fbSlamutak(
    X1 := GVL_R2.Nivaa,
    X2 := GVL_Rest.siSivState,
    XE := XE,
    SivValve1BCL := PS00_VP01.BCL,
    SivValve2BCL := PS00_VP02.BCL,
    SivValve3BCL := PS00_VP03.BCL,
    SivValve4BCL := PS00_VP04.BCL,
    ReactorValveBCL := PS02_VP01.BCL,
    ReactorValveBCH := PS02_VP01.BCH,
    PTI := GVL_Rest.Uttaksintervall,
    PTMT := GVL_Rest.MaxGangtidSlam,
    PRAntattSlamNivaa := GVL_Rest.AntattSlamNivaa);
GVL_Rest.PulseCoutner := fbSlamutak.Y;
// -------------------------------------------------------------------------------------------------------------------------------- OUTPUTS --------------------------------------------------------------------------------------------------------------------------------
// Reaktor Slamventil
// INPUTS
PS02_VP01(XGH := Sim1.BCH, XGL := Sim1.BCL, XH := fbSlamutak.YHReactorValve, XL := fbSlamutak.YLReactorValve); // SBV
Sim1(X := PS02_VP01.Y); // fbValveSim
// OUTPUTS
GVL_Outputs.PS02_VP01_Y := PS02_VP01.Y;
GVL_R2.PS02_VP01_YF := PS02_VP01.YF;
// Sivebed1
// INPUTS
PS00_VP01(XGH := Sim2.BCH, XGL := Sim2.BCL, XH := fbSlamutak.YHSivbed1Valve, XL := fbSlamutak.YLSivbed1Valve); // SBV
Sim2(X := PS00_VP01.Y); // fbValveSim
// OUTPUTS
GVL_R2.PS00_VP01_Y := PS00_VP01.Y;
GVL_R2.PS00_VP01_YF := PS00_VP01.YF;
// Sivebed2
// INPUTS
PS00_VP02(XGH := Sim3.BCH, XGL := Sim3.BCL, XH := fbSlamutak.YHSivbed2Valve, XL := fbSlamutak.YLSivbed2Valve); // SBV
Sim3(X := PS00_VP02.Y); // fbValveSim
// OUTPUTS
GVL_R2.PS00_VP02_Y := PS00_VP02.Y;
GVL_R2.PS00_VP02_YF := PS00_VP02.YF;
// Sivebed3
// INPUTS
PS00_VP03(XGH := Sim4.BCH, XGL := Sim4.BCL, XH := fbSlamutak.YHSivbed3Valve, XL := fbSlamutak.YLSivbed3Valve); // SBV
Sim4(X := PS00_VP03.Y); // fbValveSim
// OUTPUTS
GVL_R2.PS00_VP03_Y := PS00_VP03.Y;
GVL_R2.PS00_VP03_YF := PS00_VP03.YF;
// Sivebed4
// INPUTS
PS00_VP04(XGH := Sim4.BCH, XGL := Sim4.BCL, XH := fbSlamutak.YHSivbed4Valve, XL := fbSlamutak.YLSivbed4Valve); // SBV
Sim4(X := PS00_VP04.Y); // fbValveSim
// OUTPUTS
GVL_R2.PS00_VP04_Y := PS00_VP04.Y;
GVL_R2.PS00_VP04_YF := PS00_VP04.YF;

END_FUNCTION_BLOCK

// Device/Application/Simulation/Analog_I
FUNCTION_BLOCK Analog_I
VAR_INPUT
	FillLevelR	: REAL;
END_VAR
VAR_IN_OUT
	FillLevelInt	: INT;
END_VAR
VAR
	L1: LIN_TRAFO;
	L2: LIN_TRAFO;
//END_VAR
//VAR_TEMP
	Kast	: BOOL;
	temp		: REAL;
	FillV	: REAL;
END_VAR

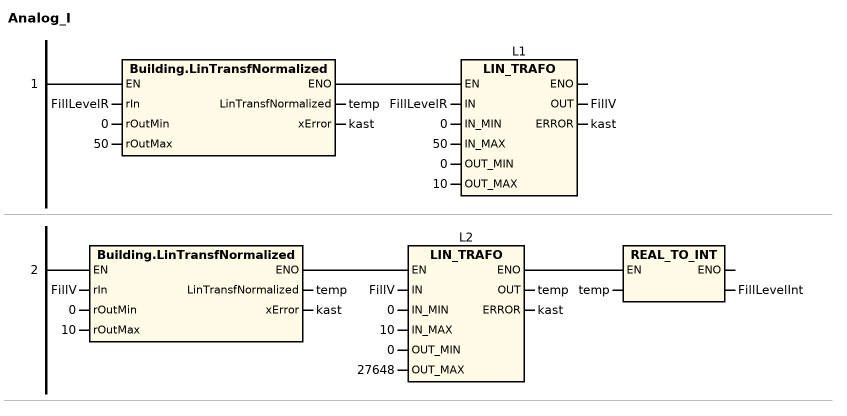
// NETWORK 1
temp := Building.LinTransfNormalized(rIn := FillLevelR, rOutMin := 0, rOutMax := 50, xError => kast);
L1(IN := FillLevelR, IN_MIN := 0, IN_MAX := 50, OUT_MIN := 0, OUT_MAX := 10, OUT => FillV, ERROR => kast); // LIN_TRAFO

// NETWORK 2
temp := Building.LinTransfNormalized(rIn := FillV, rOutMin := 0, rOutMax := 10, xError => kast);
L2(IN := FillV, IN_MIN := 0, IN_MAX := 10, OUT_MIN := 0, OUT_MAX := 27648, OUT => temp, ERROR => kast); // LIN_TRAFO
FillLevelInt := REAL_TO_INT(temp);

END_FUNCTION_BLOCK

// Device/Application/Simulation/Analog_O
FUNCTION_BLOCK Analog_O
VAR_INPUT
	PLC_Output	: INT;
END_VAR
VAR_IN_OUT
	Flow		: REAL;
END_VAR
VAR
	L1: LIN_TRAFO;
	L2: LIN_TRAFO;
//END_VAR
//VAR_TEMP
	Kast	: BOOL;
	temp		: REAL;
	PlcV	: REAL;
END_VAR

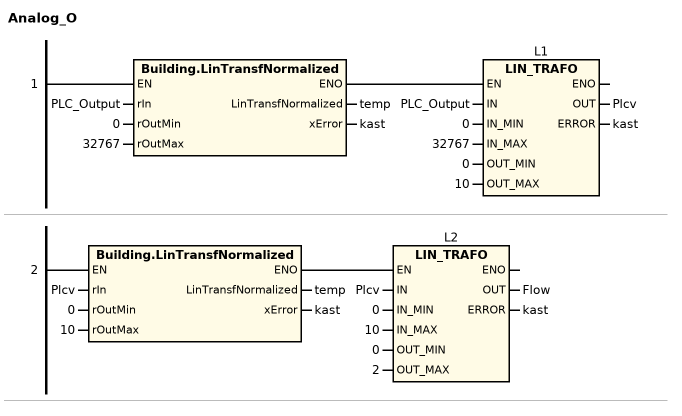
// NETWORK 1
temp := Building.LinTransfNormalized(rIn := PLC_Output, rOutMin := 0, rOutMax := 32767, xError => kast);
L1(IN := PLC_Output, IN_MIN := 0, IN_MAX := 32767, OUT_MIN := 0, OUT_MAX := 10, OUT => Plcv, ERROR => kast); // LIN_TRAFO

// NETWORK 2
temp := Building.LinTransfNormalized(rIn := Plcv, rOutMin := 0, rOutMax := 10, xError => kast);
L2(IN := Plcv, IN_MIN := 0, IN_MAX := 10, OUT_MIN := 0, OUT_MAX := 2, OUT => Flow, ERROR => kast); // LIN_TRAFO

END_FUNCTION_BLOCK

// Device/Application/Simulation/fbTankTest
FUNCTION_BLOCK fbTankTest
VAR_INPUT
	
	Start			: BOOL;	// Start av simulasjon

	StartNivaa		: REAL;	// Ved start av simulasjon kor mykje % er i tanken
	FillPerSekund	: INT;	// Tilrenning mot tank
	
	TankHoyde		: REAL;	// Dimensjonering av tank
	TankBreidde		: REAL;	// Dimensjonering av tank
	TankLengde		: REAL;	// Dimensjonering av tank
	
	TankRadius		: REAL;
	
	Drener			: BOOL; // TRUE visst tank skal drenereUT
	DrenPerSekund	: INT;	// Drenering per sekund;
	
	MotR1			: BOOL;
	Sylinder		: BOOL;
	
END_VAR
VAR_OUTPUT
	Y					: BOOL;
	OverLop				: BOOL;
	NivaBIT				: REAL;
	UtPerSekundR1		: INT;
	UtPerSekundR2		: INT;
END_VAR
VAR
	
	TankNivaa		: REAL;
	TotKubikkTank	: REAL;
	TotLTank		: REAL;
	TotProsentTank	: REAL;

	SecPuls			: fbTimer();
	L1				: LIN_TRAFO;
	
	
	sbSecPulsY		: BOOL;
	sbStart			: BOOL;
//END_VAR
//VAR_TEMP
	forkast	: BOOL;
	
	Regn	: REAL;
	
END_VAR
VAR CONSTANT
	PTD				: TIME := T#1S;	
END_VAR


SecPuls();
SecPuls.X := TRUE;
SecPuls.PTDH := PTD;

IF (Sylinder) THEN
	TotKubikkTank := TankHoyde * 3.14 * TankRadius * TankRadius;
ELSE
	TotKubikkTank := TankHoyde * TankBreidde * TankLengde;
END_IF

TotLTank	  := TotKubikkTank * 1000; // m^3 til l
Regn := StartNivaa / 100;

IF (Start AND NOT sbStart) THEN
	TankNivaa := TotLTank * Regn;
END_IF




sbStart := Start;

IF (Start) THEN
		
	IF (SecPuls.Y) THEN //AND NOT sbSecPulsY) THEN
		TankNivaa := TankNivaa + FillPerSekund;	// Adderer liter per sekund inn
		
		IF (Drener) THEN
			
			IF (MotR1) THEN
				UtPerSekundR1 := DrenPerSekund;
			ELSE
				UtPerSekundR2 := DrenPerSekund;
			END_IF
			
			Y	:= TRUE;
			TankNivaa := TankNivaa - DrenPerSekund;
		ELSE
			UtPerSekundR1 := 0;
			UtPerSekundR2 := 0;
			Y := FALSE;			
		END_IF
		
		
		SecPuls.X := FALSE;
	END_IF
	
	// Rekna ut prosent nivå i tanken	
	TotProsentTank := (TankNivaa / TotLTank) * 100;
	
	// Handle not negative TankNivaa;
	IF (TankNivaa <= 0) THEN
		DrenPerSekund := 0;
	ELSE
		DrenPersekund := DrenPerSekund;
	END_IF
	
	// Handle full
	IF (TankNivaa >= TotLTank) THEN
		TankNivaa := TotLTank;
		OverLop := TRUE;
	ELSE
		TankNivaa := TankNivaa;
		OverLop := FALSE;
	END_IF
	
	
	L1
	(
	 IN 		:= TotProsentTank,
	 IN_MIN 	:= 0,
	 IN_MAX 	:= 100,
	 OUT_MIN 	:= 5530,
	 OUT_MAX 	:= 32767,
	 OUT 		=> NivaBIT,
	 ERROR 		=> forkast
	);
ELSE
	TankNivaa := 0;
END_IF;

END_FUNCTION_BLOCK

// Device/Application/Simulation/ManualControl
FUNCTION_BLOCK ManualControl
VAR_INPUT
	PumpPower	: INT;
END_VAR	
VAR_OUTPUT
	PumpOutput	: INT;
END_VAR
VAR
	L1 : LIN_TRAFO();
//END_VAR
//VAR_TEMP
	temp	: REAL;
	kast	: BOOL;
END_VAR

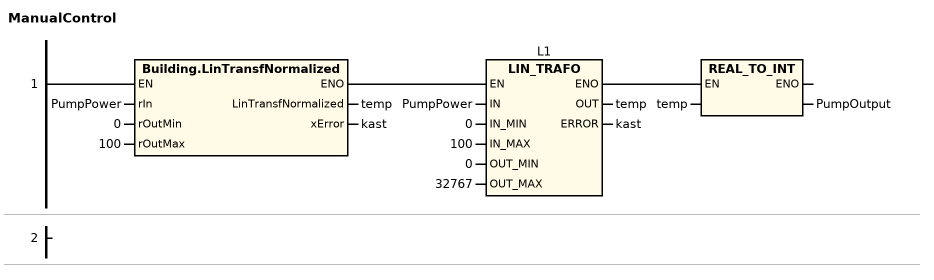
// NETWORK 1
temp := Building.LinTransfNormalized(rIn := PumpPower, rOutMin := 0, rOutMax := 100, xError => kast);
L1(IN := PumpPower, IN_MIN := 0, IN_MAX := 100, OUT_MIN := 0, OUT_MAX := 32767, OUT => temp, ERROR => kast); // LIN_TRAFO
PumpOutput := REAL_TO_INT(temp);

// NETWORK 2

END_FUNCTION_BLOCK

// Device/Application/Simulation/Simulering
PROGRAM Simulering
VAR
	Mottakstank	: fbTankTest;
	Reaktor1	: fbTankTest;
	Reaktor2	: fbTankTest;
	
	Fill		: INT;
	TimeMeter	: fbTimeMeter;
END_VAR

Mottakstank(
    Start := TRUE,
    StartNivaa := 31.6,
    FillPerSekund := Simu.FlowInlet,
    TankHoyde := 3,
    TankBreidde := 0.6,
    TankLengde := 0.6,
    Drener := GVL_Outputs.PP01_PS01_Y OR GVL_Outputs.PP02_PS01_Y,
    DrenPerSekund := 5,
    MotR1 := TRUE); // FBTANKTEST
Reaktor2(
    Start := TRUE,
    StartNivaa := 60,
    FillPerSekund := Mottakstank.UtPerSekundR2,
    TankHoyde := 0.6,
    TankRadius := 0.3,
    DrenPerSekund := Simu.FlowOutletR2,
    Sylinder := TRUE); // FBTANKTEST
// 6,3
Reaktor1(
    Start := TRUE,
    StartNivaa := 60,
    FillPerSekund := Mottakstank.UtPerSekundR1,
    TankHoyde := 0.6,
    TankRadius := 0.3,
    Drener := GVL_Outputs.TW01_VP01_Y,
    DrenPerSekund := Simu.FlowOutletR1,
    Sylinder := TRUE); // FBTANKTEST
GVL_Inputs.PP01_LT01_X := Reaktor1.NivaBIT;
GVL_Inputs.PP02_LT02_X := Reaktor2.NivaBIT;
// 3,6,6
GVL_Inputs.PP00_LT01_X := Mottakstank.NivaBIT;
TimeMeter(); // fbTimeMeter

END_PROGRAM

// Device/Application/Test_Blocks/Reaktor_2
PROGRAM Reaktor_2
VAR
//PP00_LT01	 		: MA;
END_VAR

GVL.PP00_LT01(); // MA

END_PROGRAM

// Device/Application/Simulering
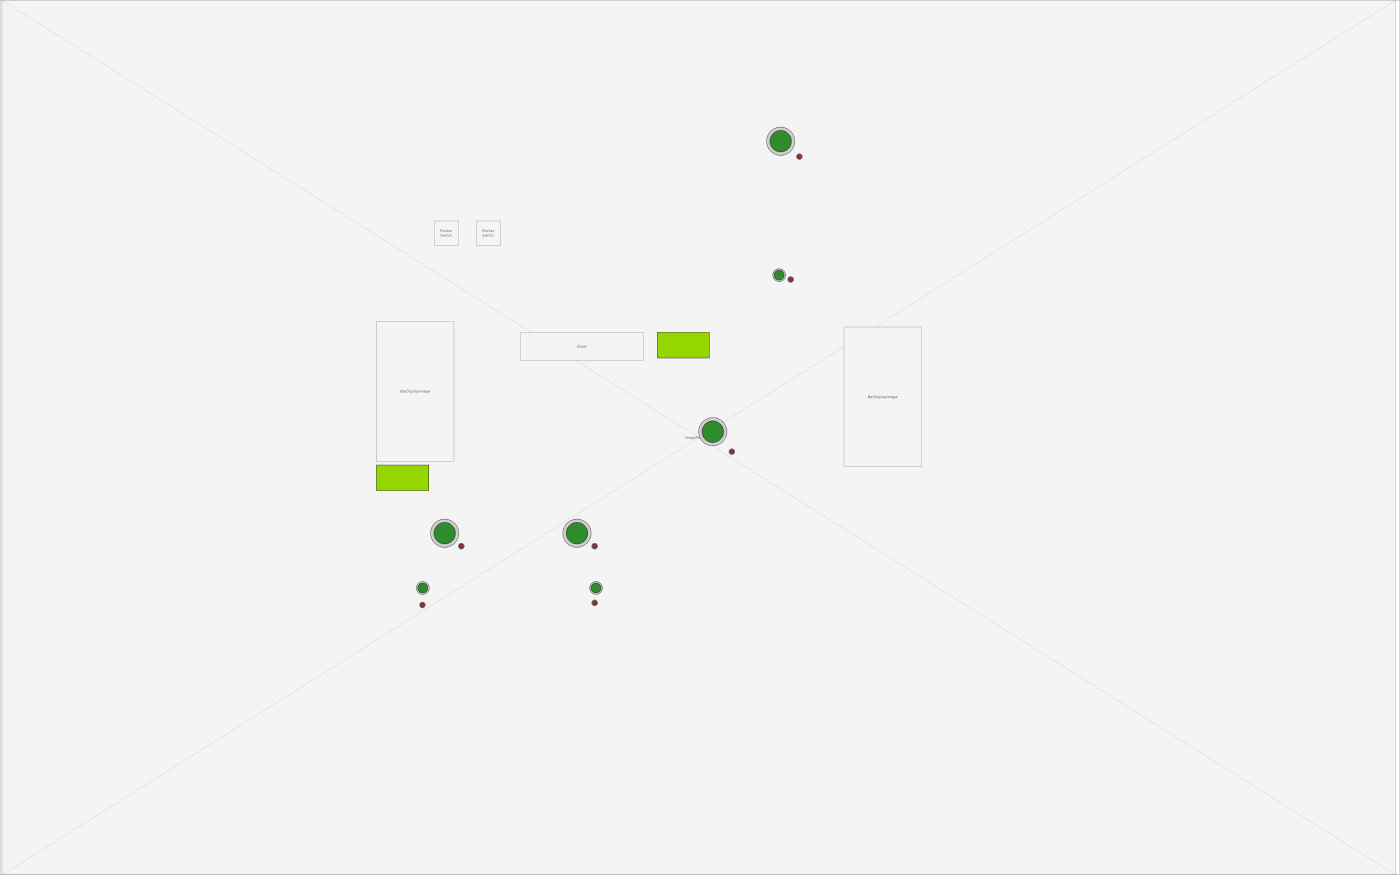
VISUALIZATION Simulering  // 4000x2500
    Image (5,0 3983x2500), image: ImagePool.P&ID
    Lamp1 (1220,1476 101x95), variable: GVL_Outputs.PP01_PS01_Y, style: Lamp-Lamp1-Green
    Lamp1 (1598,1476 101x95), variable: GVL_Outputs.PP02_PS01_Y, style: Lamp-Lamp1-Green
    RockerSwitch (1240,631 70x70), variable: GVL_Inputs.PP00_LS02_X, behaviour: TOGGLE, style: Switch-RockerSwitch-Gray
    RockerSwitch (1360,631 70x70), variable: GVL_Inputs.PP00_LS01_X, behaviour: TOGGLE, style: Switch-RockerSwitch-Gray
    BarDisplayImage (1075,918 222x400), value: Simu.MTankNivaa, style: BarDisplayImage-Gray, scale format: %.1f, scale 0..100
    Lamp1 (1186,1657 44x46), variable: GVL_Outputs.PP01_VP01_BCH, style: Lamp-Lamp1-Green
    Lamp1 (1681,1657 44x46), variable: GVL_Outputs.PP02_VP01_BCH, style: Lamp-Lamp1-Green
    Lamp1 (1689,1545 20x31), style: Lamp-Lamp1-Red
    Lamp1 (1308,1545 20x31), variable: Simu.PP01_PS01_YF, style: Lamp-Lamp1-Red
    Lamp1 (1197,1713 20x31), variable: Simu.PP01_VP01_YF, style: Lamp-Lamp1-Red
    Lamp1 (1689,1707 20x31), style: Lamp-Lamp1-Red
    Lamp1 (1986,1186 101x95), variable: GVL_Outputs.PA01_BL01_Y, style: Lamp-Lamp1-Green
    Lamp1 (2180,356 101x95), variable: GVL_Outputs.CH00_PH01_Y, style: Lamp-Lamp1-Green
    Lamp1 (2081,1275 20x31), variable: Simu.PA01_BL01_YF, style: Lamp-Lamp1-Red
    Lamp1 (2274,432 20x31), variable: Simu.CH00_PH01_YF, style: Lamp-Lamp1-Red
    Lamp1 (2204,763 44x46), variable: GVL_Outputs.TW01_VP01_BCH, style: Lamp-Lamp1-Green
    Lamp1 (2249,783 20x31), variable: Simu.TW02_VH01_YF, style: Lamp-Lamp1-Red
    BarDisplayImage (2411,934 222x400), value: Simu.R1Nivaa, style: BarDisplayImage-Gray, scale format: %.1f, scale 0..100
    Slider (1486,950 353x80), variable: Simu.FlowInlet, scale 0..50
    Rectangle (1877,949 150x74), text variable: Simu.FlowInlet
    Rectangle (1075,1328 150x74), text variable: Simu.MTankNivaa
END_VISUALIZATION

// Device/Application/Symbol
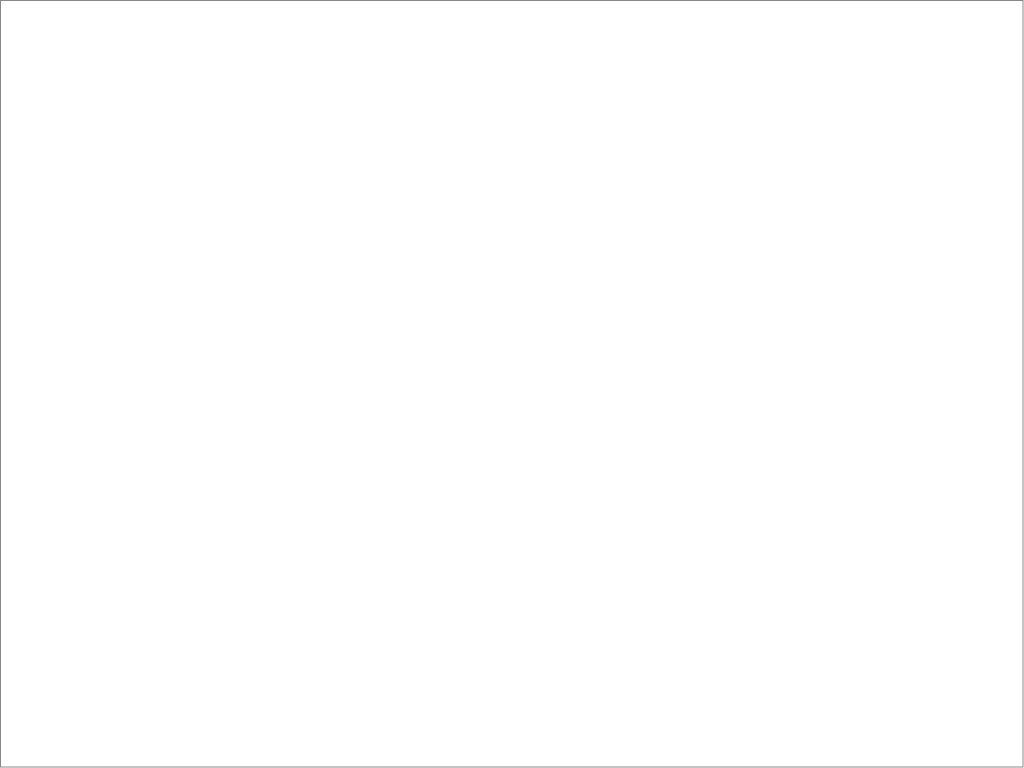
VISUALIZATION Symbol  // 1024x768
    Image (1273,344 283x238), image: VisuSymbols.Symbols.ArrowQuarterLeftRight
END_VISUALIZATION

// Device/Application/Testing
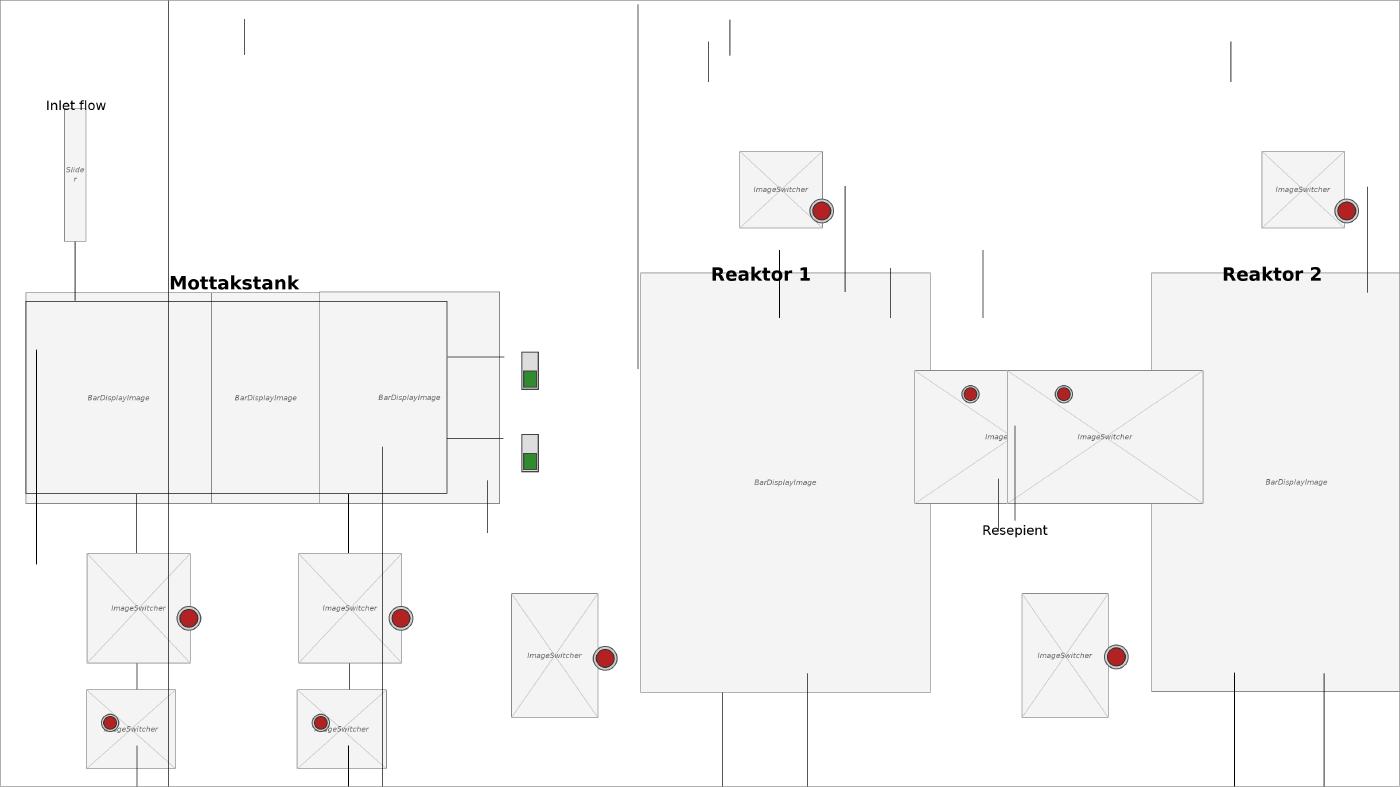
VISUALIZATION Testing  // 1920x1080
    Line (991,1087) (991,921)
    Line (479,958) (479,865)
    Line (188,958) (188,865)
    RoundedRectangle (878,401 327x522)
    BarDisplayImage (878,374 398x576), style: BarDisplayImage-Gray, scale format: %.1f, scale 0..100
    Label (969,361 150x30), "Reaktor 1"
    BarDisplayImage (237,401 255x290), style: BarDisplayImage-Gray, scale format: %.1f, scale 0..1
    BarDisplayImage (438,400 247x291), style: BarDisplayImage-Gray, scale format: %.1f, scale 0..100
    BarDisplayImage (35,401 255x290), style: BarDisplayImage-Gray, scale format: %.1f, scale 0..1
    Rectangle (35,413 578x264)
    RoundedRectangle (1579,401 327x522)
    BarDisplayImage (1579,374 398x575), style: BarDisplayImage-Gray, scale format: %.1f, scale 0..100
    Label (1670,361 150x30), "Reaktor 2"
    Label (215,373 212x30), "Mottakstank"
    ImageSwitcher (1254,508 269x183), background image: ImagePool.GreenValve, image: ImagePool.WhiteValve, behaviour: TOGGLE
    ImageSwitcher (118,946 123x109), background image: ImagePool.GreenValve90d, image: ImagePool.WhiteValve90d, behaviour: TOGGLE
    Line (187,771) (187,678)
    Line (478,771) (478,678)
    ImageSwitcher (409,759 142x151), background image: ImagePool.GreenPump90d, image: ImagePool.WhitePump90d, behaviour: TOGGLE
    ImageSwitcher (119,759 142x151), background image: ImagePool.GreenPump90d, image: ImagePool.WhitePump90d, behaviour: TOGGLE
    ImageSwitcher (407,946 123x109), background image: ImagePool.GreenValve90d, image: ImagePool.WhiteValve90d, behaviour: TOGGLE
    Line (478,1087) (478,1023)
    Line (188,1120) (188,1023)
    Line (525,1128) (525,613)
    Line (231,1162) (231,-353)
    Line (1693,1116) (1693,923)
    ImageSwitcher (1381,508 269x183), background image: ImagePool.GreenValve, image: ImagePool.WhiteValve, behaviour: TOGGLE
    Line (50,774) (50,480)
    Line (1069,436) (1069,343)
    Line (1348,436) (1348,343)
    Line (1221,436) (1221,368)
    Line (1392,714) (1392,584)
    Label (1317,713 150x30), "Resepient"
    ImageSwitcher (1014,207 114x106), background image: ImagePool.GreenPump, image: ImagePool.WhitePump, behaviour: TOGGLE
    ImageSwitcher (1730,207 114x106), background image: ImagePool.GreenPump, image: ImagePool.WhitePump, behaviour: TOGGLE
    Line (972,112) (972,57)
    Line (1688,112) (1688,57)
    Line (1159,400) (1159,255)
    Line (1875,401) (1875,256)
    ImageSwitcher (701,814 119x171), background image: ImagePool.GreenBlaser, image: ImagePool.WhiteBlaser, behaviour: TOGGLE
    ImageSwitcher (1401,814 119x171), background image: ImagePool.GreenBlaser, image: ImagePool.WhiteBlaser, behaviour: TOGGLE
    Line (669,731) (669,659)
    Line (1369,729) (1369,657)
    ImageSwitcher (1201,1364 123x109), background image: ImagePool.GreenValve90d, image: ImagePool.WhiteValve90d, behaviour: TOGGLE
    ImageSwitcher (1320,1364 123x109), background image: ImagePool.GreenValve90d, image: ImagePool.WhiteValve90d, behaviour: TOGGLE
    ImageSwitcher (1447,1364 123x109), background image: ImagePool.GreenValve90d, image: ImagePool.WhiteValve90d, behaviour: TOGGLE
    ImageSwitcher (1570,1364 123x109), background image: ImagePool.GreenValve90d, image: ImagePool.WhiteValve90d, behaviour: TOGGLE
    Line (875,506) (875,6)
    Line (1272,1377) (1272,1336)
    Line (1392,1377) (1392,1336)
    Line (1519,1376) (1519,1335)
    Line (1642,1376) (1642,1335)
    Line (1107,1105) (1107,924)
    Curve (1103,1100) (1137,1096) (1133,1132) (1117,1131) (1104,1132)
    Line (1107,1342) (1107,1127)
    ImageSwitcher (1109,1267 269x183), background image: ImagePool.GreenValve, image: ImagePool.WhiteValve, behaviour: TOGGLE
    ImageSwitcher (1668,1268 269x183), background image: ImagePool.GreenValve, image: ImagePool.WhiteValve, behaviour: TOGGLE
    Line (1816,1343) (1816,924)
    Line (335,75) (335,26)
    Line (1001,76) (1001,27)
    Line (103,412) (103,319)
    Slider (88,148 30x183), scale 0..100
    Label (13,120 183x50), "Inlet flow"
    Line (690,602) (613,602)
    Line (691,490) (614,490)
    DipSwitch (701,480 52x57), behaviour: TOGGLE, style: Switch-DipSwitch-Green
    DipSwitch (701,593 52x57), behaviour: TOGGLE, style: Switch-DipSwitch-Green
    Lamp1 (237,829 44x39), variable: GVL_Rest.PP01_PS01_YF, invisible if: NOT GVL_Rest.PP01_PS01_YF, style: Lamp-Lamp1-Red
    Lamp1 (528,829 44x39), style: Lamp-Lamp1-Red
    Lamp1 (808,884 44x39), style: Lamp-Lamp1-Red
    Lamp1 (1509,882 44x39), style: Lamp-Lamp1-Red
    Lamp1 (1105,270 44x39), style: Lamp-Lamp1-Red
    Lamp1 (1825,270 44x39), style: Lamp-Lamp1-Red
    Lamp1 (135,978 32x28), style: Lamp-Lamp1-Red
    Lamp1 (424,978 32x28), style: Lamp-Lamp1-Red
    Lamp1 (1171,1286 32x28), style: Lamp-Lamp1-Red
    Lamp1 (1218,1395 32x28), style: Lamp-Lamp1-Red
    Lamp1 (1337,1395 32x28), style: Lamp-Lamp1-Red
    Lamp1 (1464,1395 32x28), style: Lamp-Lamp1-Red
    Lamp1 (1587,1395 32x28), style: Lamp-Lamp1-Red
    Lamp1 (1729,1287 32x28), style: Lamp-Lamp1-Red
    Lamp1 (1443,527 32x28), style: Lamp-Lamp1-Red
    Lamp1 (1315,527 32x28), style: Lamp-Lamp1-Red
END_VISUALIZATION

(* text list MyStates (id | default)
  1 | Pause
  2 | Innpumping
  4 | Reaksjon
  5 | Sedimentering
  6 | Uttapping
  0 | 
   |  *)

(* text list List_alarm (id | default)
  3 | 
  2 | Anlegg i overløp
  1 | Lavt nivå mottakstank
  0 | Høgt nivå mottakstankl
   |  *)

(* text list List_Error (id | default)
  64 | Feil innløpsventil reaktor 1, safeguard mangel på tilbakemelding
  57 | Motorvern utløyst matepumpe 2
  58 | Feil innløpsventil reaktor 1, mista tilbakemelding høg
  59 | Feil innløpsventil reaktor 1, mista tilbakemelding lav
  60 | Feil innløpsventil reaktor 1, mangla tilbakemelding høg
  61 | Feil innløpsventil reaktor 1, mangla tilbakemelding lav
  62 | Innløpsventil reaktor 1 ekstern feill
  63 | Feil innløpsventil reaktor 1, safeguard blocking konflikt
  55 | Feil matepumpe 2, safeguard mangel tilbakemelding
  56 | Feil matepumpe 2, tap av aktivering
  41 | Motorvern utløyst matepumpe 1
  42 | Feil matepumpe 2, mista tilbakemeldig høg
  43 | Feil matepumpe 2, mista tilbakemelding lav
  44 | Feil matepumpe 2, mangel tilbakemelding høg
  45 | Feil matepumpe 2, mangel tilbakemelding lav
  46 | Feil matepumpe 2, ekstern feil
  47 | Feil matepumpe 2, tap av aktivering
  48 | Motorvern utløyst matepumpe 2
  49 | Feil innløpsventil reaktor 1, mista tilbakemelding høg
  50 | Feil innløpsventil reaktor 1, mista tilbakemelding lav
  51 | Feil innløpsventil reaktor 1, mangla tilbakemelding høg
  52 | Feil innløpsventil reaktor 1, mangla tilbakemelding lav
  53 | Ekstern feil
  54 | 
  40 | Feil matepumpe 1, tap av aktivering
  26 | 
  27 | 
  28 | 
  29 | 
  30 | Feil matepumpe 2, mangel tilbakemelding lav
  31 | Feil matepumpe 2, ekstern feil
  32 | Feil matepumpe 2, tap av aktivering
  33 | Motorvern utløyst matepumpe 2
  34 | Feil innløpsventil reaktor 1, mista tilbakemelding høg
  35 | Feil innløpsventil reaktor 1, mista tilbakemelding lav
  36 | Feil innløpsventil reaktor 1, mangla tilbakemelding høg
  37 | Feil innløpsventil reaktor 1, mangla tilbakemelding lav
  38 | Ekstern feil
  39 | 
  25 | 
  24 | 
  23 | 
  22 | 
  21 | 
  20 | 
  19 | 
  12 | Feil matepumpe 1, tap av aktivering
  13 | Motorvern matepumpe 1 utløyst
  14 | Feil matepumpe 2, mista tilbakemelding høg
  15 | 
  16 | 
  17 | 
  18 | 
  11 | Feil matepumpe 1, safeguard mangel tilbakemelding
  10 | Feil matepumpe 1, safeguard blocking konflikt
  9 | Feil matepumpe 1, ekstern feil
  8 | Feil matepumpe 1, mangel tilbakemelding lav
  7 | Feil matepumpe 1, mangel tilbakemelding høg
  6 | Feil matepumpe 1, mista tilbakemelding lav
  5 | Feil matepumpe 1, mista tilbakemeldig høg
  4 | Feil på trykkgivar overløp
  3 | Feil på nivåvippe høg mottakstank
  2 | Feil på nivåvippe lav mottakstank
  1 | Feil på trykkgivar mottakstank
  0 | Feilsignal grovrist
   |  *)

(* text list List_Info (id | default)
   |  *)

(* text list List_Warning (id | default)
   |  *)
